FUNCTION_BLOCK CM_Actuator2State_V2
VAR_INPUT
	
 	IN_ON : BOOL;
	Local_MODE_request : ENUM_MODE_HANDLER;
	Global_MODE_request : ENUM_MODE_HANDLER;
	
	PI_MANUAL :BOOL;
	PI_AUTO : BOOL;
	PI_HMI_HAND : BOOL;
	
	PI_AlarmHigh_Enable : BOOL;
	PI_AlarmLow_Enable : BOOL;
	
	PI_Alarm_Condition_H : BOOL;
	PI_Alarm_Condition_L : BOOL;
	
	PI_AlarmDelay_H : LREAL;
	PI_AlarmDelay_L : LREAL;
	
	PI_Alarm_Ack_H : BOOL;
	PI_Alarm_Ack_L : BOOL;
	
	PI_Interlock : BOOL;
	
	
	
END_VAR
VAR_OUTPUT
	PO_AUTO_ON :BOOL;
	PO_MANUAL_ON : BOOL;
	PO_HMI_HAND_ON : BOOL;
	
	PO_OUT_ON : BOOL;
	PO_OUT_OFF :BOOL;
	
	
	PO_ALARM_H : BOOL;
	PO_ALARM_L : BOOL;;
	
	PO_Interlocked : BOOL;
	
END_VAR
VAR
	SR_Auto: SR;
	SR_Manual : SR;
	
	Alarm_limit_Exceeded_H : BOOL;
	Alarm_limit_Exceeded_L : BOOL;
	
	Alarm_Ack_H : BOOL;
	Alarm_Ack_L : BOOL;
	
	alarmDelay_H : systemTimeDelay;
	alarmDelay_L : systemTimeDelay;
	
	MODE_HANDLER : FB_MODE_HANDLER;
END_VAR
VAR_IN_OUT
END_VAR

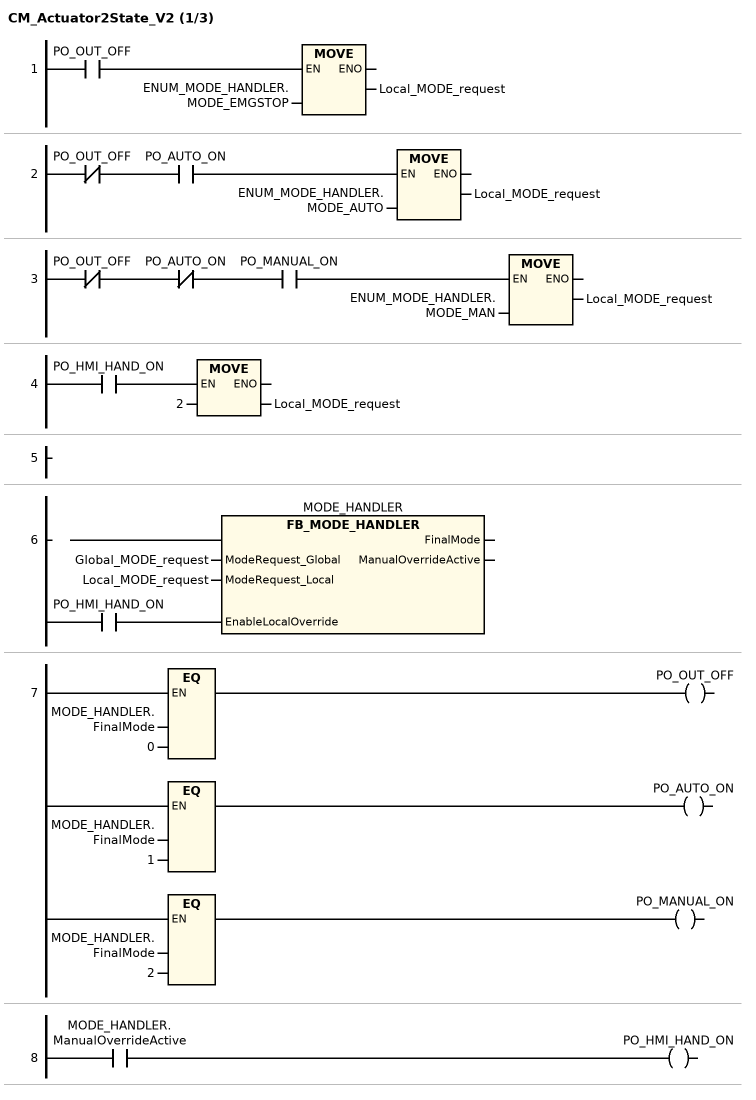
// NETWORK 1
IF PO_OUT_OFF THEN Local_MODE_request := ENUM_MODE_HANDLER.MODE_EMGSTOP; END_IF

// NETWORK 2
IF NOT PO_OUT_OFF AND PO_AUTO_ON THEN Local_MODE_request := ENUM_MODE_HANDLER.MODE_AUTO; END_IF

// NETWORK 3
IF NOT PO_OUT_OFF AND NOT PO_AUTO_ON AND PO_MANUAL_ON THEN Local_MODE_request := ENUM_MODE_HANDLER.MODE_MAN; END_IF

// NETWORK 4
IF PO_HMI_HAND_ON THEN Local_MODE_request := 2; END_IF

// NETWORK 5

// NETWORK 6
MODE_HANDLER(
    ModeRequest_Global := Global_MODE_request,
    ModeRequest_Local := Local_MODE_request,
    EnableLocalOverride := PO_HMI_HAND_ON); // FB_MODE_HANDLER

// NETWORK 7
PO_OUT_OFF := MODE_HANDLER.FinalMode = 0;
PO_AUTO_ON := MODE_HANDLER.FinalMode = 1;
PO_MANUAL_ON := MODE_HANDLER.FinalMode = 2;

// NETWORK 8
PO_HMI_HAND_ON := MODE_HANDLER.ManualOverrideActive;

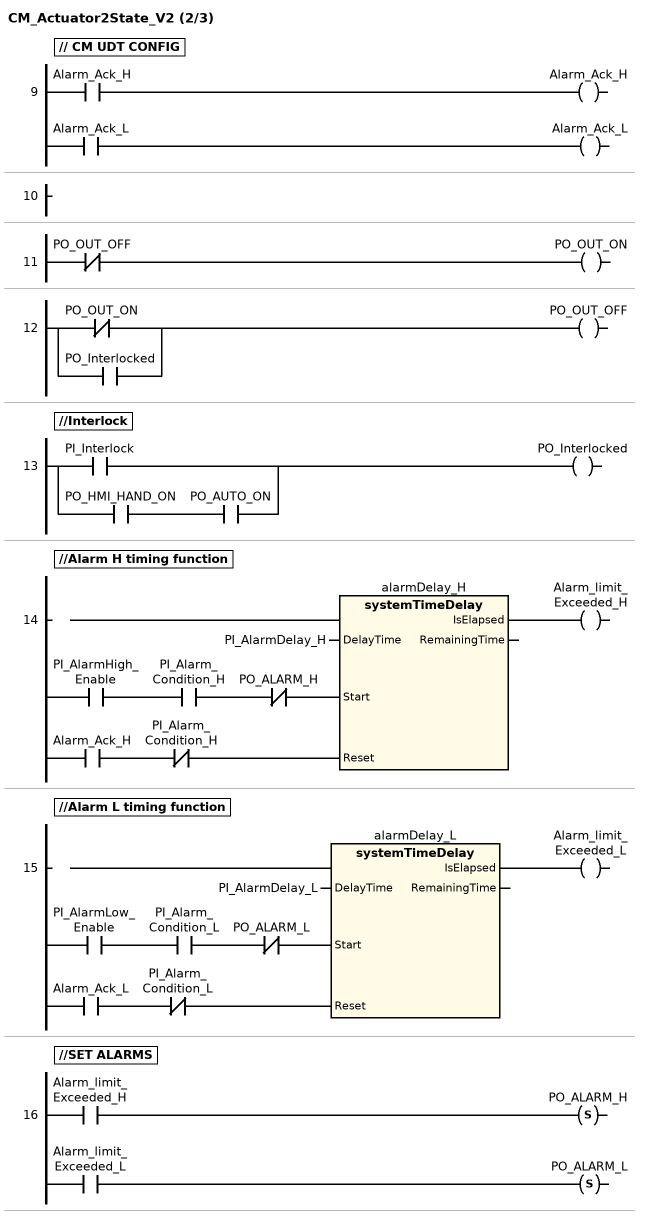
// NETWORK 9
// label: // CM UDT CONFIG
Alarm_Ack_H := Alarm_Ack_H;
Alarm_Ack_L := Alarm_Ack_L;

// NETWORK 10

// NETWORK 11
PO_OUT_ON := NOT PO_OUT_OFF;

// NETWORK 12
PO_OUT_OFF := NOT PO_OUT_ON OR PO_Interlocked;

// NETWORK 13
// label: //Interlock
PO_Interlocked := PI_Interlock OR PO_HMI_HAND_ON AND PO_AUTO_ON;

// NETWORK 14
// label: //Alarm H timing function
alarmDelay_H(
    DelayTime := PI_AlarmDelay_H,
    Start := PI_AlarmHigh_Enable AND PI_Alarm_Condition_H AND NOT PO_ALARM_H,
    Reset := Alarm_Ack_H AND NOT PI_Alarm_Condition_H); // systemTimeDelay
Alarm_limit_Exceeded_H := alarmDelay_H.IsElapsed;

// NETWORK 15
// label: //Alarm L timing function
alarmDelay_L(
    DelayTime := PI_AlarmDelay_L,
    Start := PI_AlarmLow_Enable AND PI_Alarm_Condition_L AND NOT PO_ALARM_L,
    Reset := Alarm_Ack_L AND NOT PI_Alarm_Condition_L); // systemTimeDelay
Alarm_limit_Exceeded_L := alarmDelay_L.IsElapsed;

// NETWORK 16
// label: //SET ALARMS
PO_ALARM_H S= Alarm_limit_Exceeded_H;
PO_ALARM_L S= Alarm_limit_Exceeded_L;

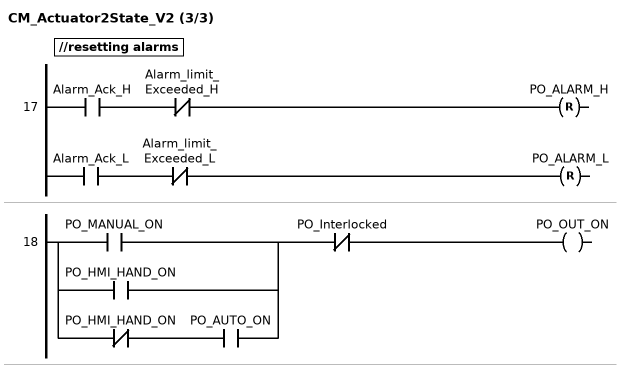
// NETWORK 17
// label: //resetting alarms
PO_ALARM_H R= Alarm_Ack_H AND NOT Alarm_limit_Exceeded_H;
PO_ALARM_L R= Alarm_Ack_L AND NOT Alarm_limit_Exceeded_L;

// NETWORK 18
PO_OUT_ON := (PO_MANUAL_ON OR PO_HMI_HAND_ON OR NOT PO_HMI_HAND_ON AND PO_AUTO_ON) AND NOT PO_Interlocked;

END_FUNCTION_BLOCK

(* stored: Version 1.1.0.1, ProductVersion 3.1.4024.13
   POU CM_Actuator2State_V2: Id {63c48792-b47e-4f9d-b254-623ecba6e2bd}, SpecialFunc None *)
